// Mitsubishi GX Developer project: パレット取り外し   PLC: Q02

PROGRAM SENSOR
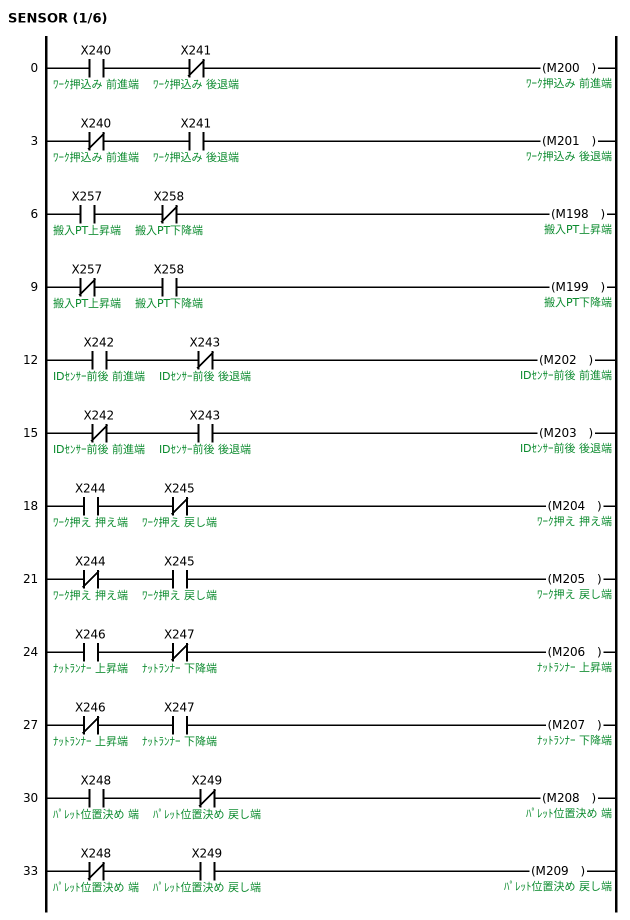
0     LD      X240  ; ﾜｰｸ押込み 前進端
      ANI     X241  ; ﾜｰｸ押込み 後退端
      OUT     M200  ; ﾜｰｸ押込み 前進端
3     LDI     X240  ; ﾜｰｸ押込み 前進端
      AND     X241  ; ﾜｰｸ押込み 後退端
      OUT     M201  ; ﾜｰｸ押込み 後退端
6     LD      X257  ; 搬入PT上昇端
      ANI     X258  ; 搬入PT下降端
      OUT     M198  ; 搬入PT上昇端
9     LDI     X257  ; 搬入PT上昇端
      AND     X258  ; 搬入PT下降端
      OUT     M199  ; 搬入PT下降端
12    LD      X242  ; IDｾﾝｻｰ前後 前進端
      ANI     X243  ; IDｾﾝｻｰ前後 後退端
      OUT     M202  ; IDｾﾝｻｰ前後 前進端
15    LDI     X242  ; IDｾﾝｻｰ前後 前進端
      AND     X243  ; IDｾﾝｻｰ前後 後退端
      OUT     M203  ; IDｾﾝｻｰ前後 後退端
18    LD      X244  ; ﾜｰｸ押え 押え端
      ANI     X245  ; ﾜｰｸ押え 戻し端
      OUT     M204  ; ﾜｰｸ押え 押え端
21    LDI     X244  ; ﾜｰｸ押え 押え端
      AND     X245  ; ﾜｰｸ押え 戻し端
      OUT     M205  ; ﾜｰｸ押え 戻し端
24    LD      X246  ; ﾅｯﾄﾗﾝﾅｰ 上昇端
      ANI     X247  ; ﾅｯﾄﾗﾝﾅｰ 下降端
      OUT     M206  ; ﾅｯﾄﾗﾝﾅｰ 上昇端
27    LDI     X246  ; ﾅｯﾄﾗﾝﾅｰ 上昇端
      AND     X247  ; ﾅｯﾄﾗﾝﾅｰ 下降端
      OUT     M207  ; ﾅｯﾄﾗﾝﾅｰ 下降端
30    LD      X248  ; ﾊﾟﾚｯﾄ位置決め 端
      ANI     X249  ; ﾊﾟﾚｯﾄ位置決め 戻し端
      OUT     M208  ; ﾊﾟﾚｯﾄ位置決め 端
33    LDI     X248  ; ﾊﾟﾚｯﾄ位置決め 端
      AND     X249  ; ﾊﾟﾚｯﾄ位置決め 戻し端
      OUT     M209  ; ﾊﾟﾚｯﾄ位置決め 戻し端
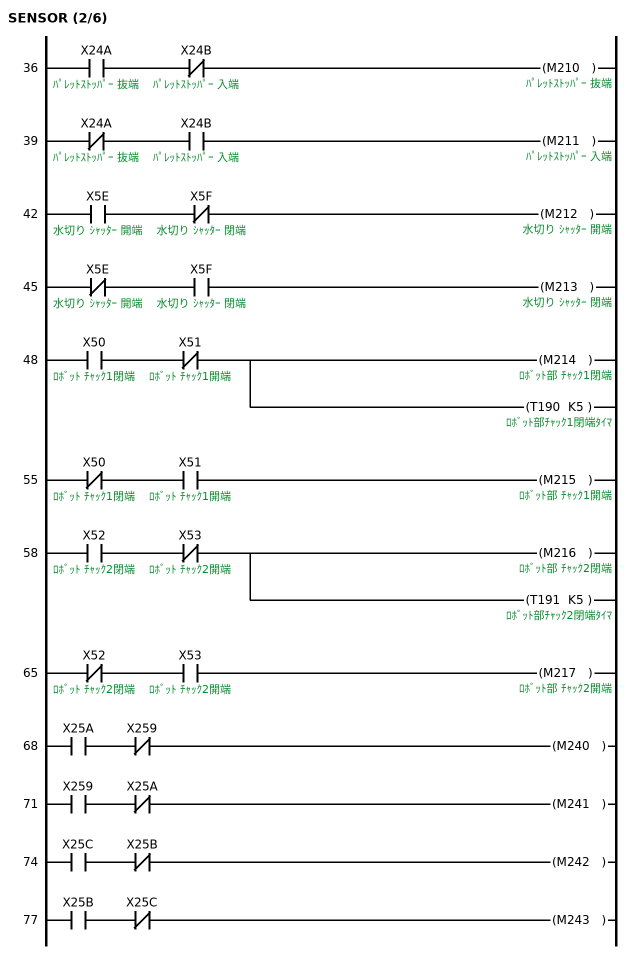
36    LD      X24A  ; ﾊﾟﾚｯﾄｽﾄｯﾊﾟｰ 抜端
      ANI     X24B  ; ﾊﾟﾚｯﾄｽﾄｯﾊﾟｰ 入端
      OUT     M210  ; ﾊﾟﾚｯﾄｽﾄｯﾊﾟｰ 抜端
39    LDI     X24A  ; ﾊﾟﾚｯﾄｽﾄｯﾊﾟｰ 抜端
      AND     X24B  ; ﾊﾟﾚｯﾄｽﾄｯﾊﾟｰ 入端
      OUT     M211  ; ﾊﾟﾚｯﾄｽﾄｯﾊﾟｰ 入端
42    LD      X5E  ; 水切り ｼｬｯﾀｰ 開端
      ANI     X5F  ; 水切り ｼｬｯﾀｰ 閉端
      OUT     M212  ; 水切り ｼｬｯﾀｰ 開端
45    LDI     X5E  ; 水切り ｼｬｯﾀｰ 開端
      AND     X5F  ; 水切り ｼｬｯﾀｰ 閉端
      OUT     M213  ; 水切り ｼｬｯﾀｰ 閉端
48    LD      X50  ; ﾛﾎﾞｯﾄ ﾁｬｯｸ1閉端
      ANI     X51  ; ﾛﾎﾞｯﾄ ﾁｬｯｸ1開端
      OUT     M214  ; ﾛﾎﾞｯﾄ部 ﾁｬｯｸ1閉端
      OUT     T190 K5  ; ﾛﾎﾞｯﾄ部ﾁｬｯｸ1閉端ﾀｲﾏ
55    LDI     X50  ; ﾛﾎﾞｯﾄ ﾁｬｯｸ1閉端
      AND     X51  ; ﾛﾎﾞｯﾄ ﾁｬｯｸ1開端
      OUT     M215  ; ﾛﾎﾞｯﾄ部 ﾁｬｯｸ1開端
58    LD      X52  ; ﾛﾎﾞｯﾄ ﾁｬｯｸ2閉端
      ANI     X53  ; ﾛﾎﾞｯﾄ ﾁｬｯｸ2開端
      OUT     M216  ; ﾛﾎﾞｯﾄ部 ﾁｬｯｸ2閉端
      OUT     T191 K5  ; ﾛﾎﾞｯﾄ部ﾁｬｯｸ2閉端ﾀｲﾏ
65    LDI     X52  ; ﾛﾎﾞｯﾄ ﾁｬｯｸ2閉端
      AND     X53  ; ﾛﾎﾞｯﾄ ﾁｬｯｸ2開端
      OUT     M217  ; ﾛﾎﾞｯﾄ部 ﾁｬｯｸ2開端
68    LD      X25A
      ANI     X259
      OUT     M240
71    LD      X259
      ANI     X25A
      OUT     M241
74    LD      X25C
      ANI     X25B
      OUT     M242
77    LD      X25B
      ANI     X25C
      OUT     M243
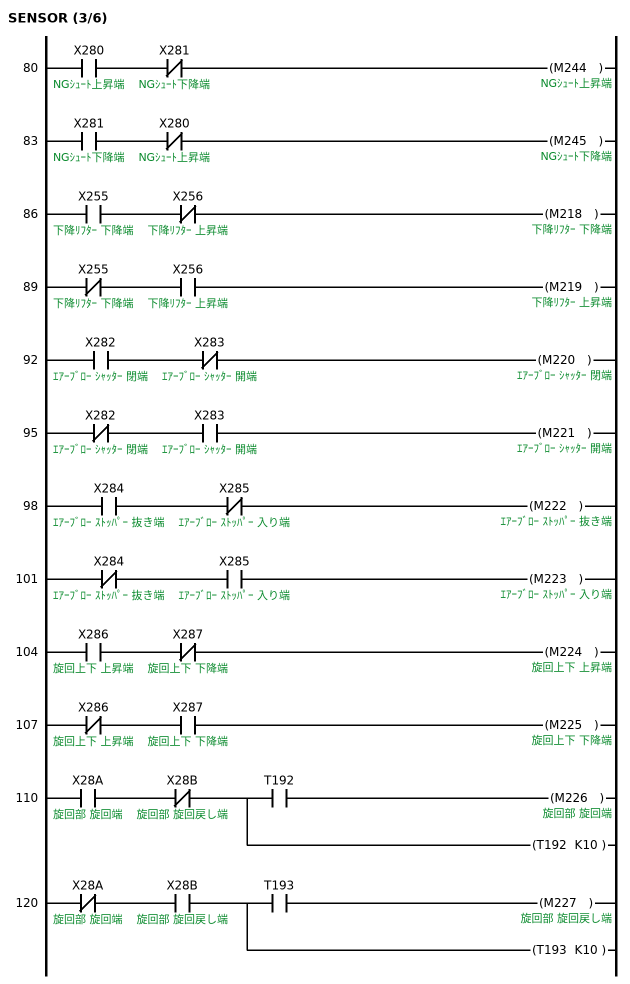
80    LD      X280  ; NGｼｭｰﾄ上昇端
      ANI     X281  ; NGｼｭｰﾄ下降端
      OUT     M244  ; NGｼｭｰﾄ上昇端
83    LD      X281  ; NGｼｭｰﾄ下降端
      ANI     X280  ; NGｼｭｰﾄ上昇端
      OUT     M245  ; NGｼｭｰﾄ下降端
86    LD      X255  ; 下降ﾘﾌﾀｰ 下降端
      ANI     X256  ; 下降ﾘﾌﾀｰ 上昇端
      OUT     M218  ; 下降ﾘﾌﾀｰ 下降端
89    LDI     X255  ; 下降ﾘﾌﾀｰ 下降端
      AND     X256  ; 下降ﾘﾌﾀｰ 上昇端
      OUT     M219  ; 下降ﾘﾌﾀｰ 上昇端
92    LD      X282  ; ｴｱｰﾌﾞﾛｰ ｼｬｯﾀｰ 閉端
      ANI     X283  ; ｴｱｰﾌﾞﾛｰ ｼｬｯﾀｰ 開端
      OUT     M220  ; ｴｱｰﾌﾞﾛｰ ｼｬｯﾀｰ 閉端
95    LDI     X282  ; ｴｱｰﾌﾞﾛｰ ｼｬｯﾀｰ 閉端
      AND     X283  ; ｴｱｰﾌﾞﾛｰ ｼｬｯﾀｰ 開端
      OUT     M221  ; ｴｱｰﾌﾞﾛｰ ｼｬｯﾀｰ 開端
98    LD      X284  ; ｴｱｰﾌﾞﾛｰ ｽﾄｯﾊﾟｰ 抜き端
      ANI     X285  ; ｴｱｰﾌﾞﾛｰ ｽﾄｯﾊﾟｰ 入り端
      OUT     M222  ; ｴｱｰﾌﾞﾛｰ ｽﾄｯﾊﾟｰ 抜き端
101   LDI     X284  ; ｴｱｰﾌﾞﾛｰ ｽﾄｯﾊﾟｰ 抜き端
      AND     X285  ; ｴｱｰﾌﾞﾛｰ ｽﾄｯﾊﾟｰ 入り端
      OUT     M223  ; ｴｱｰﾌﾞﾛｰ ｽﾄｯﾊﾟｰ 入り端
104   LD      X286  ; 旋回上下 上昇端
      ANI     X287  ; 旋回上下 下降端
      OUT     M224  ; 旋回上下 上昇端
107   LDI     X286  ; 旋回上下 上昇端
      AND     X287  ; 旋回上下 下降端
      OUT     M225  ; 旋回上下 下降端
110   LD      X28A  ; 旋回部 旋回端
      ANI     X28B  ; 旋回部 旋回戻し端
      MPS
      AND     T192
      OUT     M226  ; 旋回部 旋回端
      MPP
      OUT     T192 K10
120   LDI     X28A  ; 旋回部 旋回端
      AND     X28B  ; 旋回部 旋回戻し端
      MPS
      AND     T193
      OUT     M227  ; 旋回部 旋回戻し端
      MPP
      OUT     T193 K10
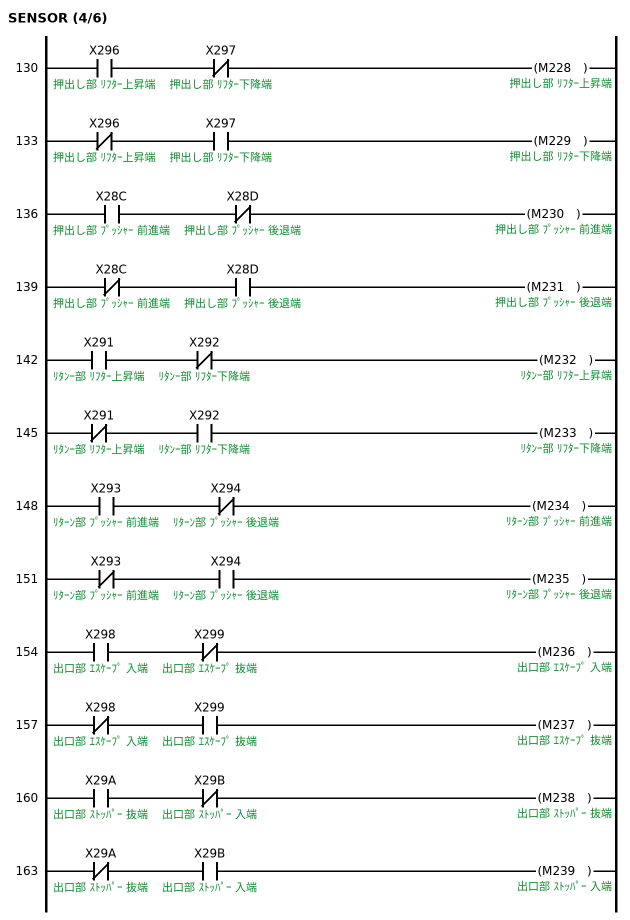
130   LD      X296  ; 押出し部 ﾘﾌﾀｰ上昇端
      ANI     X297  ; 押出し部 ﾘﾌﾀｰ下降端
      OUT     M228  ; 押出し部 ﾘﾌﾀｰ上昇端
133   LDI     X296  ; 押出し部 ﾘﾌﾀｰ上昇端
      AND     X297  ; 押出し部 ﾘﾌﾀｰ下降端
      OUT     M229  ; 押出し部 ﾘﾌﾀｰ下降端
136   LD      X28C  ; 押出し部 ﾌﾟｯｼｬｰ 前進端
      ANI     X28D  ; 押出し部 ﾌﾟｯｼｬｰ 後退端
      OUT     M230  ; 押出し部 ﾌﾟｯｼｬｰ 前進端
139   LDI     X28C  ; 押出し部 ﾌﾟｯｼｬｰ 前進端
      AND     X28D  ; 押出し部 ﾌﾟｯｼｬｰ 後退端
      OUT     M231  ; 押出し部 ﾌﾟｯｼｬｰ 後退端
142   LD      X291  ; ﾘﾀﾝｰ部 ﾘﾌﾀｰ上昇端
      ANI     X292  ; ﾘﾀﾝｰ部 ﾘﾌﾀｰ下降端
      OUT     M232  ; ﾘﾀﾝｰ部 ﾘﾌﾀｰ上昇端
145   LDI     X291  ; ﾘﾀﾝｰ部 ﾘﾌﾀｰ上昇端
      AND     X292  ; ﾘﾀﾝｰ部 ﾘﾌﾀｰ下降端
      OUT     M233  ; ﾘﾀﾝｰ部 ﾘﾌﾀｰ下降端
148   LD      X293  ; ﾘﾀｰﾝ部 ﾌﾟｯｼｬｰ 前進端
      ANI     X294  ; ﾘﾀｰﾝ部 ﾌﾟｯｼｬｰ 後退端
      OUT     M234  ; ﾘﾀｰﾝ部 ﾌﾟｯｼｬｰ 前進端
151   LDI     X293  ; ﾘﾀｰﾝ部 ﾌﾟｯｼｬｰ 前進端
      AND     X294  ; ﾘﾀｰﾝ部 ﾌﾟｯｼｬｰ 後退端
      OUT     M235  ; ﾘﾀｰﾝ部 ﾌﾟｯｼｬｰ 後退端
154   LD      X298  ; 出口部 ｴｽｹｰﾌﾟ 入端
      ANI     X299  ; 出口部 ｴｽｹｰﾌﾟ 抜端
      OUT     M236  ; 出口部 ｴｽｹｰﾌﾟ 入端
157   LDI     X298  ; 出口部 ｴｽｹｰﾌﾟ 入端
      AND     X299  ; 出口部 ｴｽｹｰﾌﾟ 抜端
      OUT     M237  ; 出口部 ｴｽｹｰﾌﾟ 抜端
160   LD      X29A  ; 出口部 ｽﾄｯﾊﾟｰ 抜端
      ANI     X29B  ; 出口部 ｽﾄｯﾊﾟｰ 入端
      OUT     M238  ; 出口部 ｽﾄｯﾊﾟｰ 抜端
163   LDI     X29A  ; 出口部 ｽﾄｯﾊﾟｰ 抜端
      AND     X29B  ; 出口部 ｽﾄｯﾊﾟｰ 入端
      OUT     M239  ; 出口部 ｽﾄｯﾊﾟｰ 入端
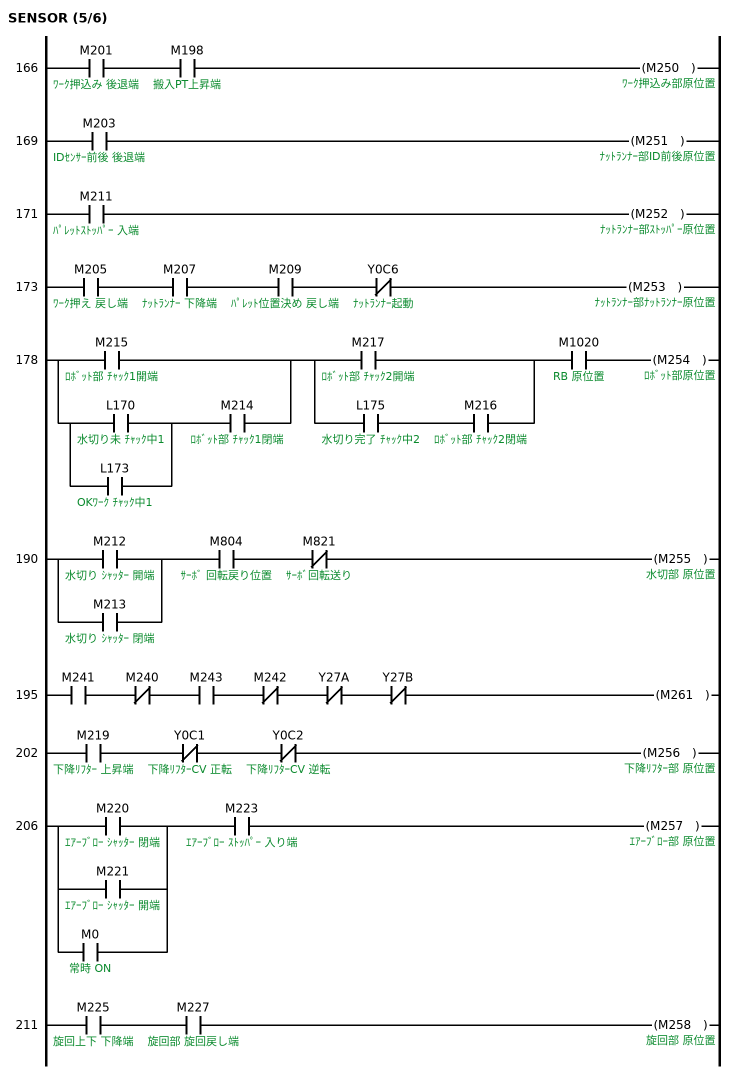
166   LD      M201  ; ﾜｰｸ押込み 後退端
      AND     M198  ; 搬入PT上昇端
      OUT     M250  ; ﾜｰｸ押込み部原位置
169   LD      M203  ; IDｾﾝｻｰ前後 後退端
      OUT     M251  ; ﾅｯﾄﾗﾝﾅｰ部ID前後原位置
171   LD      M211  ; ﾊﾟﾚｯﾄｽﾄｯﾊﾟｰ 入端
      OUT     M252  ; ﾅｯﾄﾗﾝﾅｰ部ｽﾄｯﾊﾟｰ原位置
173   LD      M205  ; ﾜｰｸ押え 戻し端
      AND     M207  ; ﾅｯﾄﾗﾝﾅｰ 下降端
      AND     M209  ; ﾊﾟﾚｯﾄ位置決め 戻し端
      ANI     Y0C6  ; ﾅｯﾄﾗﾝﾅｰ起動
      OUT     M253  ; ﾅｯﾄﾗﾝﾅｰ部ﾅｯﾄﾗﾝﾅｰ原位置
178   LD      M215  ; ﾛﾎﾞｯﾄ部 ﾁｬｯｸ1開端
      LD      L170  ; 水切り未 ﾁｬｯｸ中1
      OR      L173  ; OKﾜｰｸ ﾁｬｯｸ中1
      AND     M214  ; ﾛﾎﾞｯﾄ部 ﾁｬｯｸ1閉端
      ORB
      LD      M217  ; ﾛﾎﾞｯﾄ部 ﾁｬｯｸ2開端
      LD      L175  ; 水切り完了 ﾁｬｯｸ中2
      AND     M216  ; ﾛﾎﾞｯﾄ部 ﾁｬｯｸ2閉端
      ORB
      ANB
      AND     M1020  ; RB 原位置
      OUT     M254  ; ﾛﾎﾞｯﾄ部原位置
190   LD      M212  ; 水切り ｼｬｯﾀｰ 開端
      OR      M213  ; 水切り ｼｬｯﾀｰ 閉端
      AND     M804  ; ｻｰﾎﾞ 回転戻り位置
      ANI     M821  ; ｻｰﾎﾞ回転送り
      OUT     M255  ; 水切部 原位置
195   LD      M241
      ANI     M240
      AND     M243
      ANI     M242
      ANI     Y27A
      ANI     Y27B
      OUT     M261
202   LD      M219  ; 下降ﾘﾌﾀｰ 上昇端
      ANI     Y0C1  ; 下降ﾘﾌﾀｰCV 正転
      ANI     Y0C2  ; 下降ﾘﾌﾀｰCV 逆転
      OUT     M256  ; 下降ﾘﾌﾀｰ部 原位置
206   LD      M220  ; ｴｱｰﾌﾞﾛｰ ｼｬｯﾀｰ 閉端
      OR      M221  ; ｴｱｰﾌﾞﾛｰ ｼｬｯﾀｰ 開端
      OR      M0  ; 常時 ON
      AND     M223  ; ｴｱｰﾌﾞﾛｰ ｽﾄｯﾊﾟｰ 入り端
      OUT     M257  ; ｴｱｰﾌﾞﾛｰ部 原位置
211   LD      M225  ; 旋回上下 下降端
      AND     M227  ; 旋回部 旋回戻し端
      OUT     M258  ; 旋回部 原位置
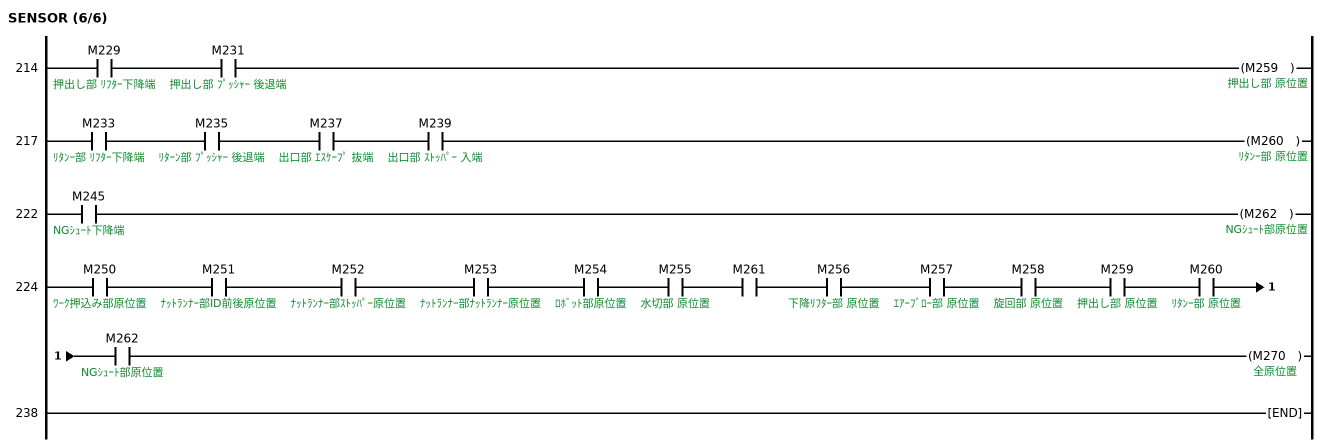
214   LD      M229  ; 押出し部 ﾘﾌﾀｰ下降端
      AND     M231  ; 押出し部 ﾌﾟｯｼｬｰ 後退端
      OUT     M259  ; 押出し部 原位置
217   LD      M233  ; ﾘﾀﾝｰ部 ﾘﾌﾀｰ下降端
      AND     M235  ; ﾘﾀｰﾝ部 ﾌﾟｯｼｬｰ 後退端
      AND     M237  ; 出口部 ｴｽｹｰﾌﾟ 抜端
      AND     M239  ; 出口部 ｽﾄｯﾊﾟｰ 入端
      OUT     M260  ; ﾘﾀﾝｰ部 原位置
222   LD      M245  ; NGｼｭｰﾄ下降端
      OUT     M262  ; NGｼｭｰﾄ部原位置
224   LD      M250  ; ﾜｰｸ押込み部原位置
      AND     M251  ; ﾅｯﾄﾗﾝﾅｰ部ID前後原位置
      AND     M252  ; ﾅｯﾄﾗﾝﾅｰ部ｽﾄｯﾊﾟｰ原位置
      AND     M253  ; ﾅｯﾄﾗﾝﾅｰ部ﾅｯﾄﾗﾝﾅｰ原位置
      AND     M254  ; ﾛﾎﾞｯﾄ部原位置
      AND     M255  ; 水切部 原位置
      AND     M261
      AND     M256  ; 下降ﾘﾌﾀｰ部 原位置
      AND     M257  ; ｴｱｰﾌﾞﾛｰ部 原位置
      AND     M258  ; 旋回部 原位置
      AND     M259  ; 押出し部 原位置
      AND     M260  ; ﾘﾀﾝｰ部 原位置
      AND     M262  ; NGｼｭｰﾄ部原位置
      OUT     M270  ; 全原位置
238   END
END_PROGRAM
